// TIA Portal V17 export
// export: Created 2025-03-07T09:17:40.5566251Z, ExportSetting WithDefaults, DisplayName Totally Integrated Automation Portal, DisplayVersion V17 Update 8, DisplayName TIA Portal Openness, DisplayVersion V17 Update 8, DisplayName TIA Portal Version Control Interface, DisplayVersion V17, DisplayName SINAMICS Startdrive Advanced, DisplayVersion V17 SP2, DisplayName SINAMICS Startdrive G110M, G120, G120C, G120D, G120P, G115D, DisplayVersion V17 SP2, DisplayName SINAMICS Startdrive G130, G150, S120, S150, SINAMICS MV, S210, DisplayVersion V17 SP2, DisplayName STEP 7 Professional, DisplayVersion V17 Update 8, DisplayName SINUMERIK ONE STEP 7 Toolbox, DisplayVersion V17 Update 12, DisplayName SINUMERIK 840D sl STEP 7 Toolbox, DisplayVersion V17 Update 12, DisplayName STEP 7 Safety, DisplayVersion V17 Update 6, DisplayName WinCC Advanced, DisplayVersion V17 Update 8
FUNCTION "FC2023_CNC_MODES_G2" : Void   // FC2023, LAD
{ S7_Optimized_Access := 'TRUE' }
VERSION : 0.1
// stored: AutoNumber false, IsIECCheckEnabled false, SetENOAutomatically false, UDAEnableTagReadback false
BEGIN

NETWORK
TITLE = ACTUAL VALUE IN WCS 0=MCS / Actual value in WCS 0=MCS
// WKS/MKS
      AN    "LBP_HMI".E_ActWCS;
      JC    M001;
      AN    "LBP_HMI".A_ActWCS;
      =     "LBP_HMI".A_ActWCS;
      CLR;
      =     "LBP_HMI".E_ActWCS;
M001: NOP   0;

REGION Network 2: MODE GROUP RESET / Mode group reset
   // BAG Reset
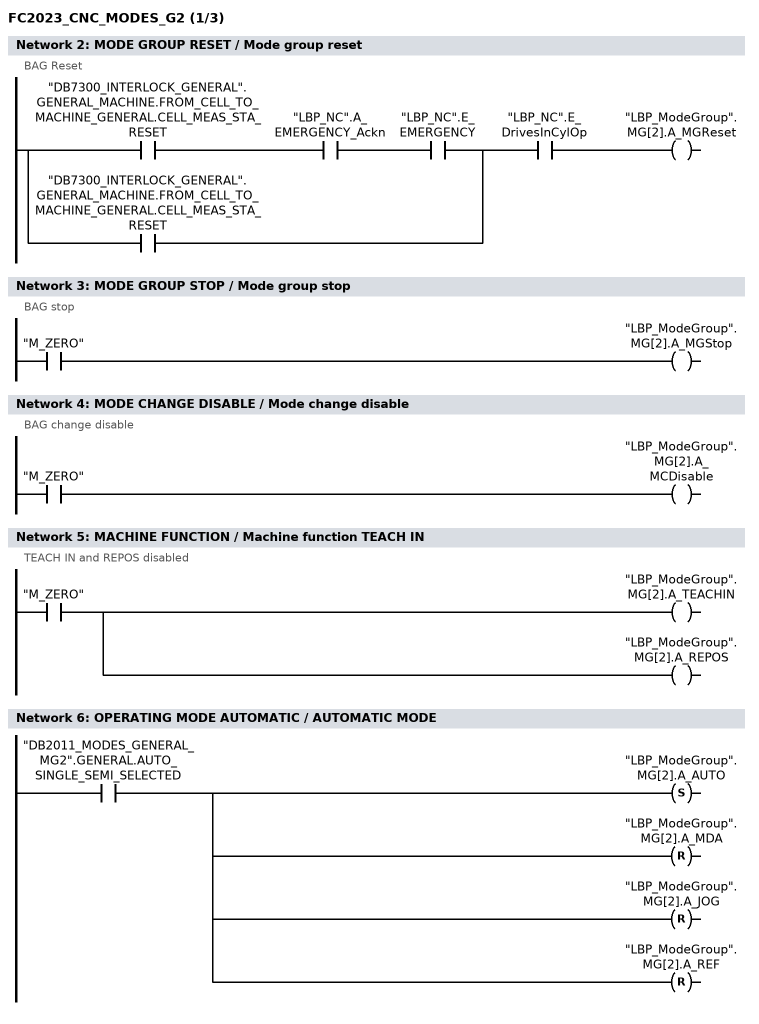
   RUNG wire#powerrail
      Contact( "DB7300_INTERLOCK_GENERAL".GENERAL_MACHINE.FROM_CELL_TO_MACHINE_GENERAL.CELL_MEAS_STA_RESET )
      Contact( "LBP_NC".A_EMERGENCY_Ackn )
      Contact( "LBP_NC".E_EMERGENCY )
      wire#w1
      Contact( "LBP_NC".E_DrivesInCylOp )
      Coil( "LBP_ModeGroup".MG[2].A_MGReset )
   END_RUNG
   RUNG wire#powerrail
      Contact( "DB7300_INTERLOCK_GENERAL".GENERAL_MACHINE.FROM_CELL_TO_MACHINE_GENERAL.CELL_MEAS_STA_RESET )
   END_RUNG wire#w1
   // the same network as SCL:
   "LBP_ModeGroup".MG[2].A_MGReset := (("DB7300_INTERLOCK_GENERAL".GENERAL_MACHINE.FROM_CELL_TO_MACHINE_GENERAL.CELL_MEAS_STA_RESET AND "LBP_NC".A_EMERGENCY_Ackn AND "LBP_NC".E_EMERGENCY) OR "DB7300_INTERLOCK_GENERAL".GENERAL_MACHINE.FROM_CELL_TO_MACHINE_GENERAL.CELL_MEAS_STA_RESET) AND "LBP_NC".E_DrivesInCylOp;
END_REGION

REGION Network 3: MODE GROUP STOP / Mode group stop
   // BAG stop
   RUNG wire#powerrail
      Contact( "M_ZERO" )
      Coil( "LBP_ModeGroup".MG[2].A_MGStop )
   END_RUNG
   // the same network as SCL:
   "LBP_ModeGroup".MG[2].A_MGStop := "M_ZERO";
END_REGION

REGION Network 4: MODE CHANGE DISABLE / Mode change disable
   // BAG change disable
   RUNG wire#powerrail
      Contact( "M_ZERO" )
      Coil( "LBP_ModeGroup".MG[2].A_MCDisable )
   END_RUNG
   // the same network as SCL:
   "LBP_ModeGroup".MG[2].A_MCDisable := "M_ZERO";
END_REGION

REGION Network 5: MACHINE FUNCTION / Machine function TEACH IN
   // TEACH IN and REPOS disabled
   RUNG wire#powerrail
      Contact( "M_ZERO" )
      wire#w1
      Coil( "LBP_ModeGroup".MG[2].A_TEACHIN )
   END_RUNG
   RUNG wire#w1
      Coil( "LBP_ModeGroup".MG[2].A_REPOS )
   END_RUNG
   // the same network as SCL:
   "LBP_ModeGroup".MG[2].A_TEACHIN := "M_ZERO";
   "LBP_ModeGroup".MG[2].A_REPOS := "M_ZERO";
END_REGION

REGION Network 6: OPERATING MODE AUTOMATIC / AUTOMATIC MODE
   RUNG wire#powerrail
      Contact( "DB2011_MODES_GENERAL_MG2".GENERAL.AUTO_SINGLE_SEMI_SELECTED )
      wire#w1
      S_Coil( "LBP_ModeGroup".MG[2].A_AUTO )
   END_RUNG
   RUNG wire#w1
      R_Coil( "LBP_ModeGroup".MG[2].A_MDA )
   END_RUNG
   RUNG wire#w1
      R_Coil( "LBP_ModeGroup".MG[2].A_JOG )
   END_RUNG
   RUNG wire#w1
      R_Coil( "LBP_ModeGroup".MG[2].A_REF )
   END_RUNG
   // the same network as SCL:
   IF "DB2011_MODES_GENERAL_MG2".GENERAL.AUTO_SINGLE_SEMI_SELECTED THEN
       "LBP_ModeGroup".MG[2].A_AUTO := TRUE;
       "LBP_ModeGroup".MG[2].A_MDA := FALSE;
       "LBP_ModeGroup".MG[2].A_JOG := FALSE;
       "LBP_ModeGroup".MG[2].A_REF := FALSE;
   END_IF;
END_REGION

REGION Network 7: OPERATING MODE MDA / MDI MODE
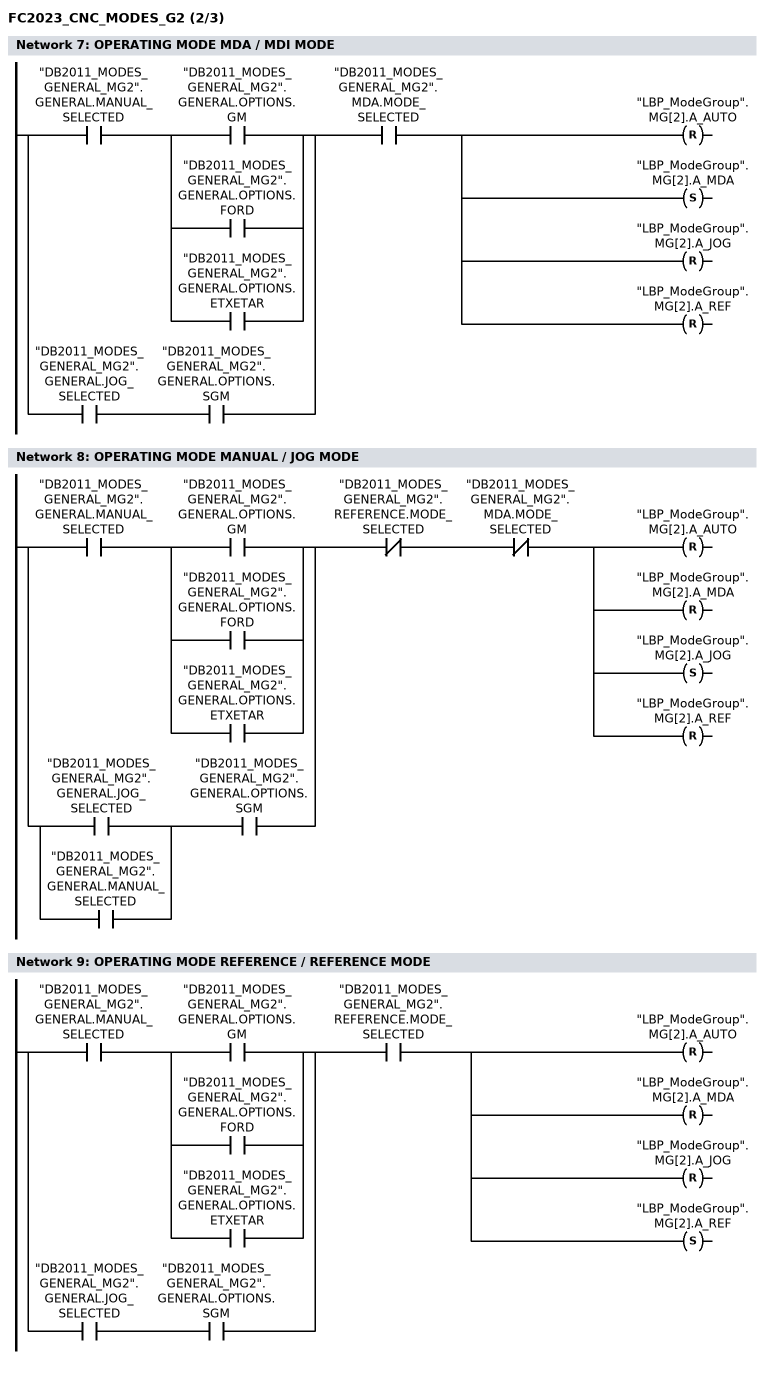
   RUNG wire#powerrail
      Contact( "DB2011_MODES_GENERAL_MG2".GENERAL.MANUAL_SELECTED )
      wire#w1
      Contact( "DB2011_MODES_GENERAL_MG2".GENERAL.OPTIONS.GM )
      wire#w2
      Contact( "DB2011_MODES_GENERAL_MG2".MDA.MODE_SELECTED )
      wire#w3
      R_Coil( "LBP_ModeGroup".MG[2].A_AUTO )
   END_RUNG
   RUNG wire#w1
      Contact( "DB2011_MODES_GENERAL_MG2".GENERAL.OPTIONS.FORD )
   END_RUNG wire#w2
   RUNG wire#w1
      Contact( "DB2011_MODES_GENERAL_MG2".GENERAL.OPTIONS.ETXETAR )
   END_RUNG wire#w2
   RUNG wire#powerrail
      Contact( "DB2011_MODES_GENERAL_MG2".GENERAL.JOG_SELECTED )
      Contact( "DB2011_MODES_GENERAL_MG2".GENERAL.OPTIONS.SGM )
   END_RUNG wire#w2
   RUNG wire#w3
      S_Coil( "LBP_ModeGroup".MG[2].A_MDA )
   END_RUNG
   RUNG wire#w3
      R_Coil( "LBP_ModeGroup".MG[2].A_JOG )
   END_RUNG
   RUNG wire#w3
      R_Coil( "LBP_ModeGroup".MG[2].A_REF )
   END_RUNG
   // the same network as SCL:
   IF (("DB2011_MODES_GENERAL_MG2".GENERAL.MANUAL_SELECTED AND ("DB2011_MODES_GENERAL_MG2".GENERAL.OPTIONS.GM OR "DB2011_MODES_GENERAL_MG2".GENERAL.OPTIONS.FORD OR "DB2011_MODES_GENERAL_MG2".GENERAL.OPTIONS.ETXETAR)) OR ("DB2011_MODES_GENERAL_MG2".GENERAL.JOG_SELECTED AND "DB2011_MODES_GENERAL_MG2".GENERAL.OPTIONS.SGM)) AND "DB2011_MODES_GENERAL_MG2".MDA.MODE_SELECTED THEN
       "LBP_ModeGroup".MG[2].A_AUTO := FALSE;
       "LBP_ModeGroup".MG[2].A_MDA := TRUE;
       "LBP_ModeGroup".MG[2].A_JOG := FALSE;
       "LBP_ModeGroup".MG[2].A_REF := FALSE;
   END_IF;
END_REGION

REGION Network 8: OPERATING MODE MANUAL / JOG MODE
   RUNG wire#powerrail
      Contact( "DB2011_MODES_GENERAL_MG2".GENERAL.MANUAL_SELECTED )
      wire#w1
      Contact( "DB2011_MODES_GENERAL_MG2".GENERAL.OPTIONS.GM )
      wire#w2
      I_Contact( "DB2011_MODES_GENERAL_MG2".REFERENCE.MODE_SELECTED )
      I_Contact( "DB2011_MODES_GENERAL_MG2".MDA.MODE_SELECTED )
      wire#w4
      R_Coil( "LBP_ModeGroup".MG[2].A_AUTO )
   END_RUNG
   RUNG wire#w1
      Contact( "DB2011_MODES_GENERAL_MG2".GENERAL.OPTIONS.FORD )
   END_RUNG wire#w2
   RUNG wire#w1
      Contact( "DB2011_MODES_GENERAL_MG2".GENERAL.OPTIONS.ETXETAR )
   END_RUNG wire#w2
   RUNG wire#powerrail
      Contact( "DB2011_MODES_GENERAL_MG2".GENERAL.JOG_SELECTED )
      wire#w3
      Contact( "DB2011_MODES_GENERAL_MG2".GENERAL.OPTIONS.SGM )
   END_RUNG wire#w2
   RUNG wire#powerrail
      Contact( "DB2011_MODES_GENERAL_MG2".GENERAL.MANUAL_SELECTED )
   END_RUNG wire#w3
   RUNG wire#w4
      R_Coil( "LBP_ModeGroup".MG[2].A_MDA )
   END_RUNG
   RUNG wire#w4
      S_Coil( "LBP_ModeGroup".MG[2].A_JOG )
   END_RUNG
   RUNG wire#w4
      R_Coil( "LBP_ModeGroup".MG[2].A_REF )
   END_RUNG
   // the same network as SCL:
   IF (("DB2011_MODES_GENERAL_MG2".GENERAL.MANUAL_SELECTED AND ("DB2011_MODES_GENERAL_MG2".GENERAL.OPTIONS.GM OR "DB2011_MODES_GENERAL_MG2".GENERAL.OPTIONS.FORD OR "DB2011_MODES_GENERAL_MG2".GENERAL.OPTIONS.ETXETAR)) OR (("DB2011_MODES_GENERAL_MG2".GENERAL.JOG_SELECTED OR "DB2011_MODES_GENERAL_MG2".GENERAL.MANUAL_SELECTED) AND "DB2011_MODES_GENERAL_MG2".GENERAL.OPTIONS.SGM)) AND NOT "DB2011_MODES_GENERAL_MG2".REFERENCE.MODE_SELECTED AND NOT "DB2011_MODES_GENERAL_MG2".MDA.MODE_SELECTED THEN
       "LBP_ModeGroup".MG[2].A_AUTO := FALSE;
       "LBP_ModeGroup".MG[2].A_MDA := FALSE;
       "LBP_ModeGroup".MG[2].A_JOG := TRUE;
       "LBP_ModeGroup".MG[2].A_REF := FALSE;
   END_IF;
END_REGION

REGION Network 9: OPERATING MODE REFERENCE / REFERENCE MODE
   RUNG wire#powerrail
      Contact( "DB2011_MODES_GENERAL_MG2".GENERAL.MANUAL_SELECTED )
      wire#w1
      Contact( "DB2011_MODES_GENERAL_MG2".GENERAL.OPTIONS.GM )
      wire#w2
      Contact( "DB2011_MODES_GENERAL_MG2".REFERENCE.MODE_SELECTED )
      wire#w3
      R_Coil( "LBP_ModeGroup".MG[2].A_AUTO )
   END_RUNG
   RUNG wire#w1
      Contact( "DB2011_MODES_GENERAL_MG2".GENERAL.OPTIONS.FORD )
   END_RUNG wire#w2
   RUNG wire#w1
      Contact( "DB2011_MODES_GENERAL_MG2".GENERAL.OPTIONS.ETXETAR )
   END_RUNG wire#w2
   RUNG wire#powerrail
      Contact( "DB2011_MODES_GENERAL_MG2".GENERAL.JOG_SELECTED )
      Contact( "DB2011_MODES_GENERAL_MG2".GENERAL.OPTIONS.SGM )
   END_RUNG wire#w2
   RUNG wire#w3
      R_Coil( "LBP_ModeGroup".MG[2].A_MDA )
   END_RUNG
   RUNG wire#w3
      R_Coil( "LBP_ModeGroup".MG[2].A_JOG )
   END_RUNG
   RUNG wire#w3
      S_Coil( "LBP_ModeGroup".MG[2].A_REF )
   END_RUNG
   // the same network as SCL:
   IF (("DB2011_MODES_GENERAL_MG2".GENERAL.MANUAL_SELECTED AND ("DB2011_MODES_GENERAL_MG2".GENERAL.OPTIONS.GM OR "DB2011_MODES_GENERAL_MG2".GENERAL.OPTIONS.FORD OR "DB2011_MODES_GENERAL_MG2".GENERAL.OPTIONS.ETXETAR)) OR ("DB2011_MODES_GENERAL_MG2".GENERAL.JOG_SELECTED AND "DB2011_MODES_GENERAL_MG2".GENERAL.OPTIONS.SGM)) AND "DB2011_MODES_GENERAL_MG2".REFERENCE.MODE_SELECTED THEN
       "LBP_ModeGroup".MG[2].A_AUTO := FALSE;
       "LBP_ModeGroup".MG[2].A_MDA := FALSE;
       "LBP_ModeGroup".MG[2].A_JOG := FALSE;
       "LBP_ModeGroup".MG[2].A_REF := TRUE;
   END_IF;
END_REGION

REGION Network 10: OPERATING MODE NO MODE / NO REFERENCE MODE
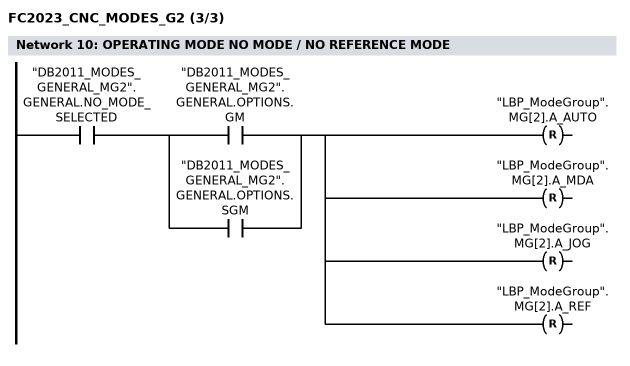
   RUNG wire#powerrail
      Contact( "DB2011_MODES_GENERAL_MG2".GENERAL.NO_MODE_SELECTED )
      wire#w1
      Contact( "DB2011_MODES_GENERAL_MG2".GENERAL.OPTIONS.GM )
      wire#w2
      R_Coil( "LBP_ModeGroup".MG[2].A_AUTO )
   END_RUNG
   RUNG wire#w1
      Contact( "DB2011_MODES_GENERAL_MG2".GENERAL.OPTIONS.SGM )
   END_RUNG wire#w2
   RUNG wire#w2
      R_Coil( "LBP_ModeGroup".MG[2].A_MDA )
   END_RUNG
   RUNG wire#w2
      R_Coil( "LBP_ModeGroup".MG[2].A_JOG )
   END_RUNG
   RUNG wire#w2
      R_Coil( "LBP_ModeGroup".MG[2].A_REF )
   END_RUNG
   // the same network as SCL:
   IF "DB2011_MODES_GENERAL_MG2".GENERAL.NO_MODE_SELECTED AND ("DB2011_MODES_GENERAL_MG2".GENERAL.OPTIONS.GM OR "DB2011_MODES_GENERAL_MG2".GENERAL.OPTIONS.SGM) THEN
       "LBP_ModeGroup".MG[2].A_AUTO := FALSE;
       "LBP_ModeGroup".MG[2].A_MDA := FALSE;
       "LBP_ModeGroup".MG[2].A_JOG := FALSE;
       "LBP_ModeGroup".MG[2].A_REF := FALSE;
   END_IF;
END_REGION
END_FUNCTION
